// Mitsubishi GX Works2 project: 0625(타이머_순차점등)   PLC: Q02/Q02H

PROGRAM MAIN
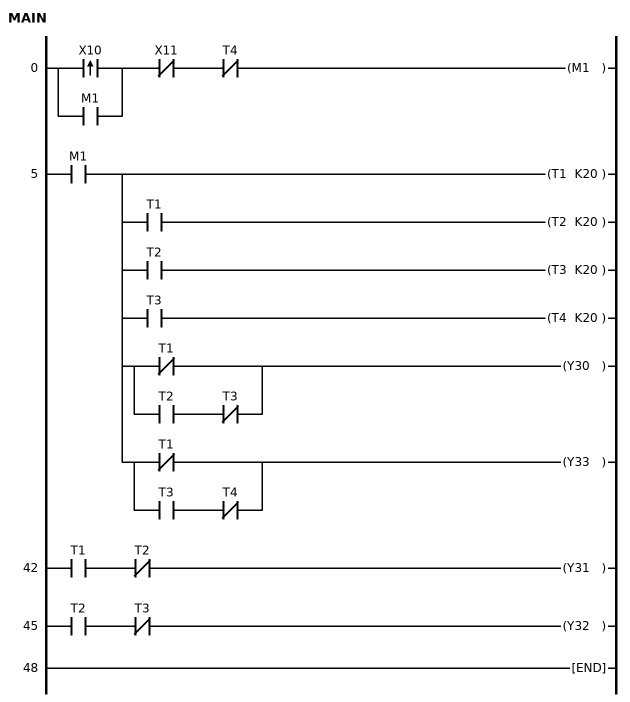
0     LDP     X10
      OR      M1
      ANI     X11
      ANI     T4
      OUT     M1
5     LD      M1
      OUT     T1 K20
      MPS
      AND     T1
      OUT     T2 K20
      MRD
      AND     T2
      OUT     T3 K20
      MRD
      AND     T3
      OUT     T4 K20
      MRD
      LDI     T1
      LD      T2
      ANI     T3
      ORB
      ANB
      OUT     Y30
      MPP
      LDI     T1
      LD      T3
      ANI     T4
      ORB
      ANB
      OUT     Y33
42    LD      T1
      ANI     T2
      OUT     Y31
45    LD      T2
      ANI     T3
      OUT     Y32
48    END
END_PROGRAM
